% RSLogix 500 project I2P Job 14 Alexander_Loynd.RSS, saved by version 10.00.00.00 %
PROJECT "ML06A"    % processor: Bul.1763 MicroLogix 1100 Series B %

PROGRAM FILES
  LAD 2   13 rungs

DATA FILES
  O0 OUTPUT  4 elements
  I1 INPUT  6 elements
  S2 STATUS  66 elements
  B3 BINARY  1 elements
  T4 TIMER  1 elements
  C5 COUNTER  1 elements
  R6 CONTROL  1 elements
  N7 INTEGER  1 elements
  F8 FLOAT  1 elements

LADDER 2
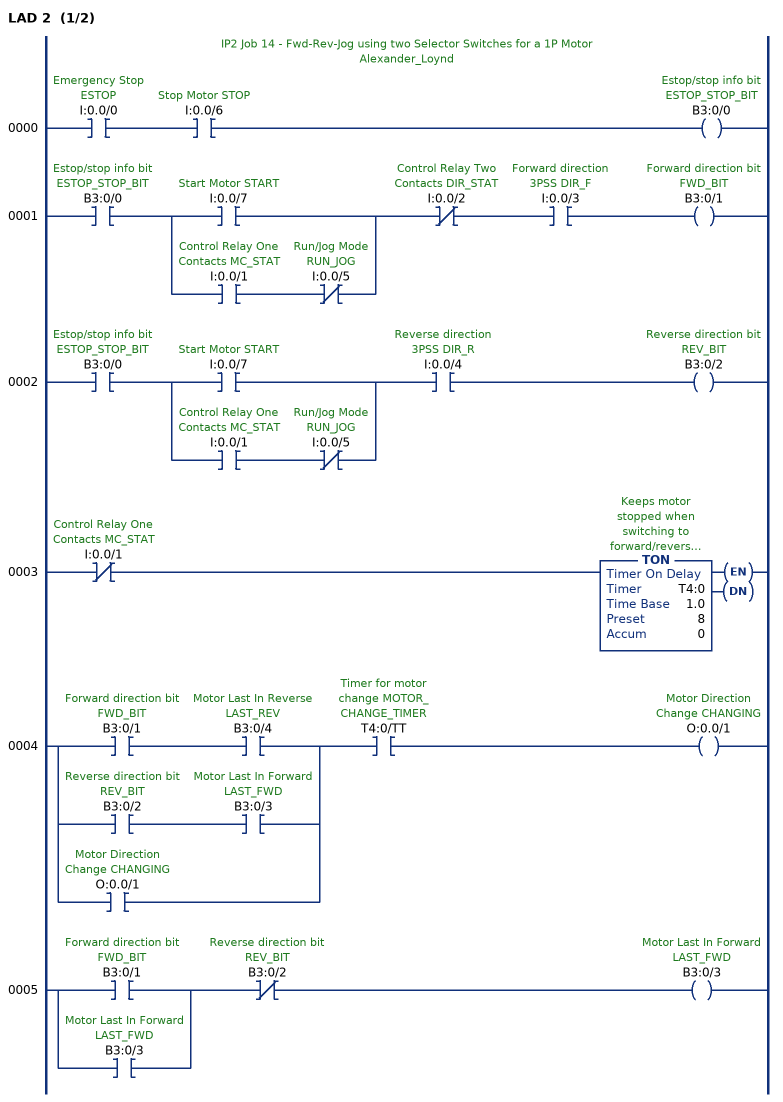
% Rung: 0 %
% IP2 Job 14 - Fwd-Rev-Jog using two Selector Switches for a 1P Motor
% Alexander_Loynd %
SOR XIC I:0.0/0 XIC I:0.0/6 OTE B3:0/0 EOR
%   I:0.0/0  ESTOP  "Emergency Stop" %
%   I:0.0/6  STOP  "Stop Motor" %
%   B3:0/0  ESTOP_STOP_BIT  "Estop/stop info bit" %
% Rung: 1 %
SOR XIC B3:0/0 BST XIC I:0.0/7 NXB XIC I:0.0/1 XIO I:0.0/5 BND XIO I:0.0/2 XIC I:0.0/3 OTE B3:0/1 EOR
%   B3:0/0  ESTOP_STOP_BIT  "Estop/stop info bit" %
%   I:0.0/7  START  "Start Motor" %
%   I:0.0/1  MC_STAT  "Control Relay One Contacts" %
%   I:0.0/5  RUN_JOG  "Run/Jog Mode" %
%   I:0.0/2  DIR_STAT  "Control Relay Two Contacts" %
%   I:0.0/3  DIR_F  "Forward direction 3PSS" %
%   B3:0/1  FWD_BIT  "Forward direction bit" %
% Rung: 2 %
SOR XIC B3:0/0 BST XIC I:0.0/7 NXB XIC I:0.0/1 XIO I:0.0/5 BND XIC I:0.0/4 OTE B3:0/2 EOR
%   B3:0/0  ESTOP_STOP_BIT  "Estop/stop info bit" %
%   I:0.0/7  START  "Start Motor" %
%   I:0.0/1  MC_STAT  "Control Relay One Contacts" %
%   I:0.0/5  RUN_JOG  "Run/Jog Mode" %
%   I:0.0/4  DIR_R  "Reverse direction 3PSS" %
%   B3:0/2  REV_BIT  "Reverse direction bit" %
% Rung: 3 %
SOR XIO I:0.0/1 TON T4:0 1.0 8 0 EOR
%   I:0.0/1  MC_STAT  "Control Relay One Contacts" %
%   T4:0  MTR_DELAY  "Keeps motor stopped when switching to forward/reverse" %
% Rung: 4 %
SOR BST XIC B3:0/1 XIC B3:0/4 NXB XIC B3:0/2 XIC B3:0/3 NXB XIC O:0.0/1 BND XIC T4:0/TT OTE O:0.0/1 EOR
%   B3:0/1  FWD_BIT  "Forward direction bit" %
%   B3:0/4  LAST_REV  "Motor Last In Reverse" %
%   B3:0/2  REV_BIT  "Reverse direction bit" %
%   B3:0/3  LAST_FWD  "Motor Last In Forward" %
%   O:0.0/1  CHANGING  "Motor Direction Change" %
%   T4:0/TT  MOTOR_CHANGE_TIMER  "Timer for motor change" %
% Rung: 5 %
SOR BST XIC B3:0/1 NXB XIC B3:0/3 BND XIO B3:0/2 OTE B3:0/3 EOR
%   B3:0/1  FWD_BIT  "Forward direction bit" %
%   B3:0/3  LAST_FWD  "Motor Last In Forward" %
%   B3:0/2  REV_BIT  "Reverse direction bit" %

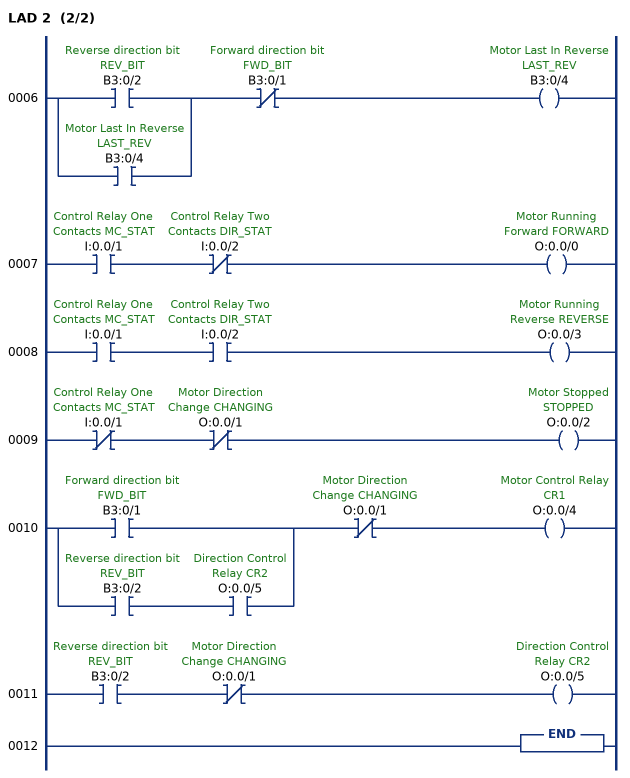
% Rung: 6 %
SOR BST XIC B3:0/2 NXB XIC B3:0/4 BND XIO B3:0/1 OTE B3:0/4 EOR
%   B3:0/2  REV_BIT  "Reverse direction bit" %
%   B3:0/4  LAST_REV  "Motor Last In Reverse" %
%   B3:0/1  FWD_BIT  "Forward direction bit" %
% Rung: 7 %
SOR XIC I:0.0/1 XIO I:0.0/2 OTE O:0.0/0 EOR
%   I:0.0/1  MC_STAT  "Control Relay One Contacts" %
%   I:0.0/2  DIR_STAT  "Control Relay Two Contacts" %
%   O:0.0/0  FORWARD  "Motor Running Forward" %
% Rung: 8 %
SOR XIC I:0.0/1 XIC I:0.0/2 OTE O:0.0/3 EOR
%   I:0.0/1  MC_STAT  "Control Relay One Contacts" %
%   I:0.0/2  DIR_STAT  "Control Relay Two Contacts" %
%   O:0.0/3  REVERSE  "Motor Running Reverse" %
% Rung: 9 %
SOR XIO I:0.0/1 XIO O:0.0/1 OTE O:0.0/2 EOR
%   I:0.0/1  MC_STAT  "Control Relay One Contacts" %
%   O:0.0/1  CHANGING  "Motor Direction Change" %
%   O:0.0/2  STOPPED  "Motor Stopped" %
% Rung: 10 %
SOR BST XIC B3:0/1 NXB XIC B3:0/2 XIC O:0.0/5 BND XIO O:0.0/1 OTE O:0.0/4 EOR
%   B3:0/1  FWD_BIT  "Forward direction bit" %
%   B3:0/2  REV_BIT  "Reverse direction bit" %
%   O:0.0/5  CR2  "Direction Control Relay" %
%   O:0.0/1  CHANGING  "Motor Direction Change" %
%   O:0.0/4  CR1  "Motor Control Relay" %
% Rung: 11 %
SOR XIC B3:0/2 XIO O:0.0/1 OTE O:0.0/5 EOR
%   B3:0/2  REV_BIT  "Reverse direction bit" %
%   O:0.0/1  CHANGING  "Motor Direction Change" %
%   O:0.0/5  CR2  "Direction Control Relay" %
% Rung: 12 %
SOR END EOR

OTHER DOCUMENTED ADDRESSES
  I:0.0/8  REV  "Start Motor in reverse"
  PB1  "Start Motor"

DATA TABLE (non-zero values as saved)
DATA T4
% .PRE .ACC %
% T4:0 % 8 0
